// TIA Portal V17 export
// export: Created 2025-05-22T06:00:28.3771667Z, ExportSetting WithDefaults, DisplayName Totally Integrated Automation Portal, DisplayVersion V17 Update 8, DisplayName TIA Portal Openness, DisplayVersion V17 Update 8, DisplayName TIA Portal Version Control Interface, DisplayVersion V17, DisplayName SINAMICS Startdrive Advanced, DisplayVersion V17 SP2, DisplayName SINAMICS Startdrive G110M, G120, G120C, G120D, G120P, G115D, DisplayVersion V17 SP2, DisplayName SINAMICS Startdrive G130, G150, S120, S150, SINAMICS MV, S210, DisplayVersion V17 SP2, DisplayName STEP 7 Professional, DisplayVersion V17 Update 8, DisplayName SINUMERIK ONE STEP 7 Toolbox, DisplayVersion V17 Update 12, DisplayName SINUMERIK ONE PLC Basic Program Plus, DisplayVersion V17 Update 12, DisplayName SINUMERIK 840D sl STEP 7 Toolbox, DisplayVersion V17 Update 12, DisplayName STEP 7 Safety, DisplayVersion V17 Update 6, DisplayName WinCC Advanced, DisplayVersion V17 Update 8
FUNCTION "FC1401_UTILITY_SKIDS" : Void   // FC1401, LAD
{ S7_Optimized_Access := 'TRUE' }
VERSION : 0.1
// stored: AutoNumber false, IsIECCheckEnabled false, SetENOAutomatically false, UDAEnableTagReadback false
   VAR CONSTANT
      FC_NUMBER : DInt := 1401;
   END_VAR
   VAR_TEMP   // added for the SCL form of the ladder/FBD networks
      _w1 : Bool;
      _w2 : Bool;
   END_VAR
BEGIN

REGION Network 1: <<<<<<<<<<<<<<<<<<<< PNEUMATIC SYSTEM >>>>>>>>>>>>>>>>>>>>
END_REGION

REGION Network 2: CALL FB1401 PNEUMATIC SYSTEM
   // 2#0000_0001 OPTIONS 0 BIT 0 PRESSURE PRESENT OPTION
   // 2#0000_0010 OPTIONS 0 BIT 1 CONNECTION SENSOR 1 OPTION
   // 2#0000_0100 OPTIONS 0 BIT 2 CONNECTION SENSOR 2 OPTION
   // 2#0000_1000 OPTIONS 0 BIT 3 DRIVE UNBLOCKED OPTION
   // 2#0001_0000 OPTIONS 0 BIT 4 PRESSURIZED OPTION
   // 2#0010_0000 OPTIONS 0 BIT 5 UNIT 01 GRIPPER PRESSURIZED OPTION
   // 2#0100_0000 OPTIONS 0 BIT 6 UNIT 01 LABERINT PRESSURIZED OPTION
   // 2#1000_0000 OPTIONS 0 BIT 7 UNIT 01 UPPER TABLE PRESSURIZED OPTION
   // 
   // 2#0000_0001 OPTIONS 1 BIT 0 UNIT 01 LOWER TABLE PRESSURIZED OPTION
   // 2#0000_0010 OPTIONS 1 BIT 1 UNIT 01 AXIS X CART PRESSURIZED OPTION
   // 2#0000_0100 OPTIONS 1 BIT 2 UNIT 01 STATION 3 MEASURMENT UNIT PRESSURIZED OPTION
   // 2#0000_1000 OPTIONS 1 BIT 3 UNIT 01 STATION 4 MEASURMENT UNIT PRESSURIZED OPTION
   // 2#0001_0000 OPTIONS 1 BIT 4 UNIT 02 GRIPPER PRESSURIZEDPRESSURIZED OPTION
   // 2#0010_0000 OPTIONS 1 BIT 5 UNIT 02 LABERINT PRESSURIZED OPTION
   // 2#0100_0000 OPTIONS 1 BIT 6 UNIT 02 UPPER TABLE PRESSURIZED OPTION
   // 2#1000_0000 OPTIONS 1 BIT 7 UNIT 02 LOWER TABLE PRESSURIZED OPTION
   // 
   // 2#0000_0001 OPTIONS 2 BIT 0 UNIT 02 AXIS X CART PRESSURIZED OPTION
   // 2#0000_0010 OPTIONS 2 BIT 1 UNIT 02 STATION 3 MEASURMENT UNIT PRESSURIZED OPTION
   // 2#0000_0100 OPTIONS 2 BIT 2 UNIT 02 STATION 4 MEASURMENT UNIT PRESSURIZED OPTION
   // 2#0000_1000 OPTIONS 2 BIT 3 INPUT FLOW  OPTION
   // 2#0001_0000 OPTIONS 2 BIT 4 INPUT TEMPERATURE OPTION
   // 2#0010_0000 OPTIONS 2 BIT 5 SPARE OPTION
   // 2#0100_0000 OPTIONS 2 BIT 6 SPARE OPTION
   // 2#1000_0000 OPTIONS 2 BIT 7 SPARE OPTION
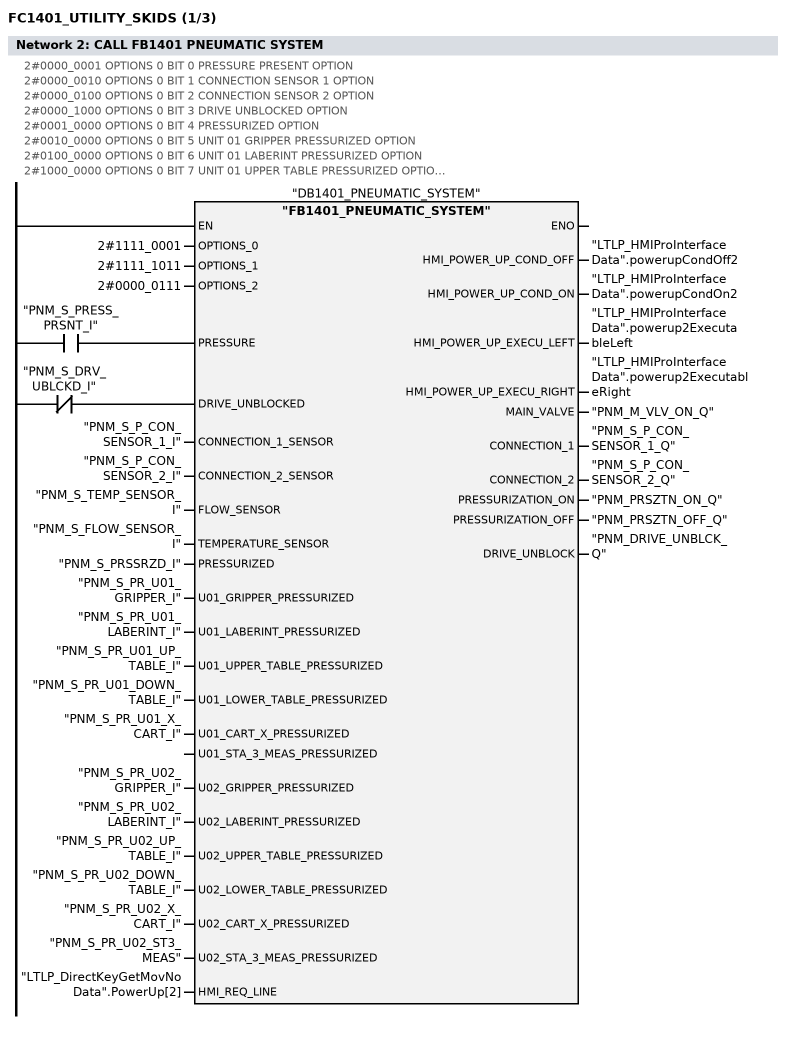
   RUNG wire#powerrail
      "DB1401_PNEUMATIC_SYSTEM"(PRESSURE := wire#w1, DRIVE_UNBLOCKED := wire#w2, OPTIONS_0 := 2#1111_0001, OPTIONS_1 := 2#1111_1011, OPTIONS_2 := 2#0000_0111, CONNECTION_1_SENSOR := "PNM_S_P_CON_SENSOR_1_I", CONNECTION_2_SENSOR := "PNM_S_P_CON_SENSOR_2_I", FLOW_SENSOR := "PNM_S_TEMP_SENSOR_I", TEMPERATURE_SENSOR := "PNM_S_FLOW_SENSOR_I", PRESSURIZED := "PNM_S_PRSSRZD_I", U01_GRIPPER_PRESSURIZED := "PNM_S_PR_U01_GRIPPER_I", U01_LABERINT_PRESSURIZED := "PNM_S_PR_U01_LABERINT_I", U01_UPPER_TABLE_PRESSURIZED := "PNM_S_PR_U01_UP_TABLE_I", U01_LOWER_TABLE_PRESSURIZED := "PNM_S_PR_U01_DOWN_TABLE_I", U01_CART_X_PRESSURIZED := "PNM_S_PR_U01_X_CART_I", U01_STA_3_MEAS_PRESSURIZED :=, U02_GRIPPER_PRESSURIZED := "PNM_S_PR_U02_GRIPPER_I", U02_LABERINT_PRESSURIZED := "PNM_S_PR_U02_LABERINT_I", U02_UPPER_TABLE_PRESSURIZED := "PNM_S_PR_U02_UP_TABLE_I", U02_LOWER_TABLE_PRESSURIZED := "PNM_S_PR_U02_DOWN_TABLE_I", U02_CART_X_PRESSURIZED := "PNM_S_PR_U02_X_CART_I", U02_STA_3_MEAS_PRESSURIZED := "PNM_S_PR_U02_ST3_MEAS", HMI_REQ_LINE := "LTLP_DirectKeyGetMovNoData".PowerUp[2], HMI_POWER_UP_COND_OFF => "LTLP_HMIProInterfaceData".powerupCondOff2, HMI_POWER_UP_COND_ON => "LTLP_HMIProInterfaceData".powerupCondOn2, HMI_POWER_UP_EXECU_LEFT => "LTLP_HMIProInterfaceData".powerup2ExecutableLeft, HMI_POWER_UP_EXECU_RIGHT => "LTLP_HMIProInterfaceData".powerup2ExecutableRight, MAIN_VALVE => "PNM_M_VLV_ON_Q", CONNECTION_1 => "PNM_S_P_CON_SENSOR_1_Q", CONNECTION_2 => "PNM_S_P_CON_SENSOR_2_Q", PRESSURIZATION_ON => "PNM_PRSZTN_ON_Q", PRESSURIZATION_OFF => "PNM_PRSZTN_OFF_Q", DRIVE_UNBLOCK => "PNM_DRIVE_UNBLCK_Q")
   END_RUNG
   RUNG wire#powerrail
      Contact( "PNM_S_PRESS_PRSNT_I" )
   END_RUNG wire#w1
   RUNG wire#powerrail
      I_Contact( "PNM_S_DRV_UBLCKD_I" )
   END_RUNG wire#w2
   // the same network as SCL:
   "DB1401_PNEUMATIC_SYSTEM"(OPTIONS_0 := 2#1111_0001,   // "FB1401_PNEUMATIC_SYSTEM"
                           OPTIONS_1 := 2#1111_1011,
                           OPTIONS_2 := 2#0000_0111,
                           PRESSURE := "PNM_S_PRESS_PRSNT_I",
                           DRIVE_UNBLOCKED := NOT "PNM_S_DRV_UBLCKD_I",
                           CONNECTION_1_SENSOR := "PNM_S_P_CON_SENSOR_1_I",
                           CONNECTION_2_SENSOR := "PNM_S_P_CON_SENSOR_2_I",
                           FLOW_SENSOR := "PNM_S_TEMP_SENSOR_I",
                           TEMPERATURE_SENSOR := "PNM_S_FLOW_SENSOR_I",
                           PRESSURIZED := "PNM_S_PRSSRZD_I",
                           U01_GRIPPER_PRESSURIZED := "PNM_S_PR_U01_GRIPPER_I",
                           U01_LABERINT_PRESSURIZED := "PNM_S_PR_U01_LABERINT_I",
                           U01_UPPER_TABLE_PRESSURIZED := "PNM_S_PR_U01_UP_TABLE_I",
                           U01_LOWER_TABLE_PRESSURIZED := "PNM_S_PR_U01_DOWN_TABLE_I",
                           U01_CART_X_PRESSURIZED := "PNM_S_PR_U01_X_CART_I",
                           U02_GRIPPER_PRESSURIZED := "PNM_S_PR_U02_GRIPPER_I",
                           U02_LABERINT_PRESSURIZED := "PNM_S_PR_U02_LABERINT_I",
                           U02_UPPER_TABLE_PRESSURIZED := "PNM_S_PR_U02_UP_TABLE_I",
                           U02_LOWER_TABLE_PRESSURIZED := "PNM_S_PR_U02_DOWN_TABLE_I",
                           U02_CART_X_PRESSURIZED := "PNM_S_PR_U02_X_CART_I",
                           U02_STA_3_MEAS_PRESSURIZED := "PNM_S_PR_U02_ST3_MEAS",
                           HMI_REQ_LINE := "LTLP_DirectKeyGetMovNoData".PowerUp[2],
                           HMI_POWER_UP_COND_OFF => "LTLP_HMIProInterfaceData".powerupCondOff2,
                           HMI_POWER_UP_COND_ON => "LTLP_HMIProInterfaceData".powerupCondOn2,
                           HMI_POWER_UP_EXECU_LEFT => "LTLP_HMIProInterfaceData".powerup2ExecutableLeft,
                           HMI_POWER_UP_EXECU_RIGHT => "LTLP_HMIProInterfaceData".powerup2ExecutableRight,
                           MAIN_VALVE => "PNM_M_VLV_ON_Q",
                           CONNECTION_1 => "PNM_S_P_CON_SENSOR_1_Q",
                           CONNECTION_2 => "PNM_S_P_CON_SENSOR_2_Q",
                           PRESSURIZATION_ON => "PNM_PRSZTN_ON_Q",
                           PRESSURIZATION_OFF => "PNM_PRSZTN_OFF_Q",
                           DRIVE_UNBLOCK => "PNM_DRIVE_UNBLCK_Q");
END_REGION

REGION Network 3: <<<<<<<<<<<<<<<<<<<< LUBRICATION SYSTEM >>>>>>>>>>>>>>>>>>>>
END_REGION

REGION Network 4: CALL FB1421 PROGRESSIVE LUBRICATION WITH GREASE
   // 2#0000_0001 OPTIONS 0 BIT 0 CIRCUIT BREAKER OPTION
   // 2#0000_0010 OPTIONS 0 BIT 1 LOW LEVEL ALARM OPTION
   // 2#0000_0100 OPTIONS 0 BIT 2 OVERPRESSURE ALARM OPTION
   // 2#0000_1000 OPTIONS 0 BIT 3 LUBRICATION BY TIME VALVE 1 AXIS X OPTION
   // 2#0001_0000 OPTIONS 0 BIT 4 LUBRICATION BY TIME VALVE 2 AXIS Z OPTION
   // 2#0010_0000 OPTIONS 0 BIT 5 LUBRICATION BY TIME VALVE 3 TURN UNIT OPTION
   // 2#0100_0000 OPTIONS 0 BIT 6 LUBRICATION BY TIME VALVE 4 OPTION
   // 2#1000_0000 OPTIONS 0 BIT 7 LUBRICATION DONE VALVE 1  AXIS X OPTION
   // 
   // 2#0000_0001 OPTIONS 1 BIT 0 LUBRICATION DONE VALVE 2 AXIS Z OPTION
   // 2#0000_0010 OPTIONS 1 BIT 1 LUBRICATION DONE VALVE 3 TURN UNIT OPTION
   // 2#0000_0100 OPTIONS 1 BIT 2 LUBRICATION DONE VALVE 4 OPTION
   // 2#0000_1000 OPTIONS 1 BIT 3 LUBRICATION DONE VALVE 5 OPTION
   // 2#0001_0000 OPTIONS 1 BIT 4 LUBRICATION DONE VALVE 6 OPTION
   // 2#0010_0000 OPTIONS 1 BIT 5 LUBRICATION DONE VALVE 7 OPTION
   // 2#0100_0000 OPTIONS 1 BIT 6 LUBRICATION DONE VALVE 8 OPTION
   // 2#1000_0000 OPTIONS 1 BIT 7 LUBRICATION DONE VALVE 9 OPTION
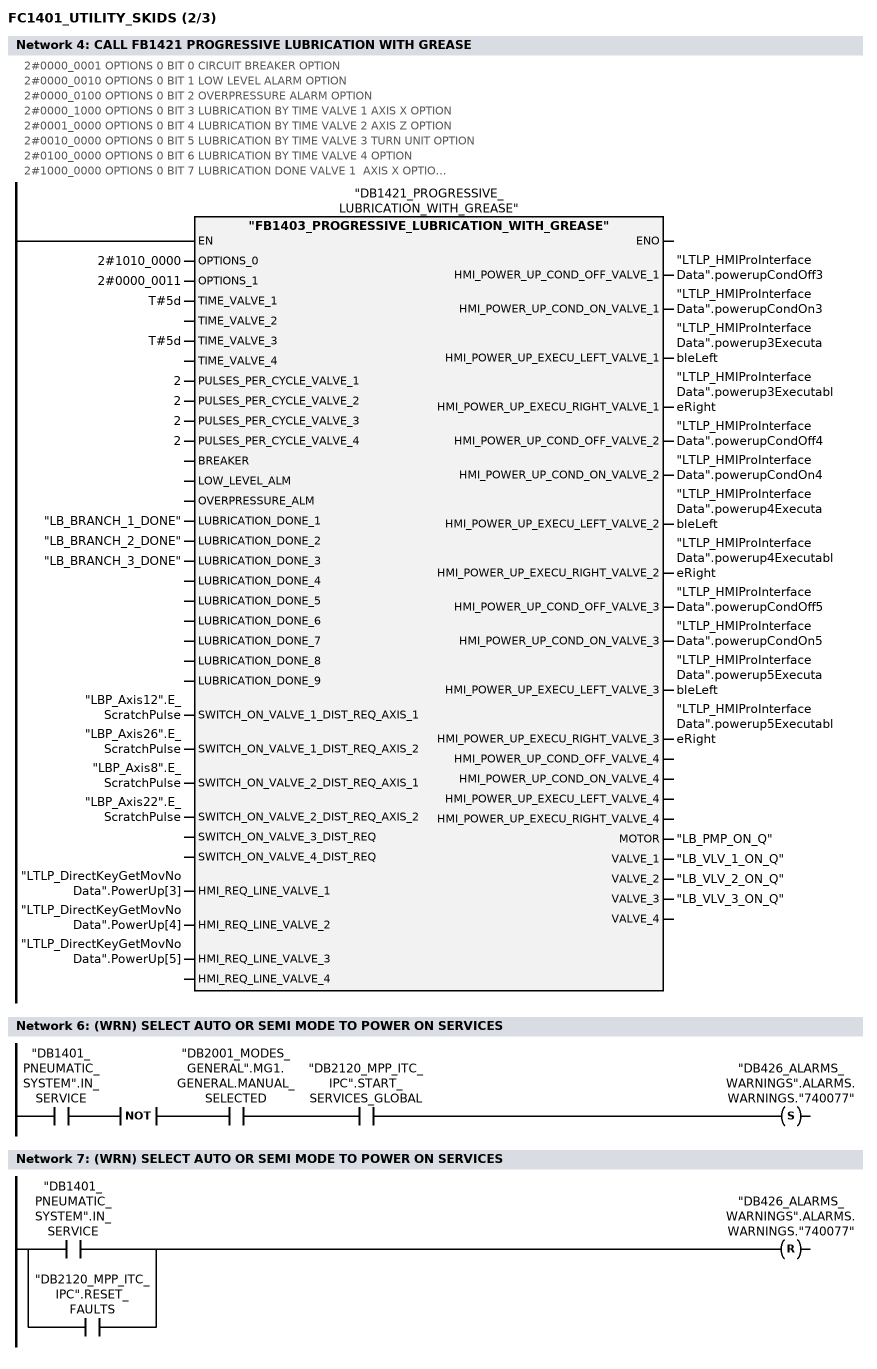
   RUNG wire#powerrail
      "DB1421_PROGRESSIVE_LUBRICATION_WITH_GREASE"(OPTIONS_0 := 2#1010_0000, OPTIONS_1 := 2#0000_0011, TIME_VALVE_1 := T#5d, TIME_VALVE_2 :=, TIME_VALVE_3 := T#5d, TIME_VALVE_4 :=, PULSES_PER_CYCLE_VALVE_1 := 2, PULSES_PER_CYCLE_VALVE_2 := 2, PULSES_PER_CYCLE_VALVE_3 := 2, PULSES_PER_CYCLE_VALVE_4 := 2, BREAKER :=, LOW_LEVEL_ALM :=, OVERPRESSURE_ALM :=, LUBRICATION_DONE_1 := "LB_BRANCH_1_DONE", LUBRICATION_DONE_2 := "LB_BRANCH_2_DONE", LUBRICATION_DONE_3 := "LB_BRANCH_3_DONE", LUBRICATION_DONE_4 :=, LUBRICATION_DONE_5 :=, LUBRICATION_DONE_6 :=, LUBRICATION_DONE_7 :=, LUBRICATION_DONE_8 :=, LUBRICATION_DONE_9 :=, SWITCH_ON_VALVE_1_DIST_REQ_AXIS_1 := "LBP_Axis12".E_ScratchPulse, SWITCH_ON_VALVE_1_DIST_REQ_AXIS_2 := "LBP_Axis26".E_ScratchPulse, SWITCH_ON_VALVE_2_DIST_REQ_AXIS_1 := "LBP_Axis8".E_ScratchPulse, SWITCH_ON_VALVE_2_DIST_REQ_AXIS_2 := "LBP_Axis22".E_ScratchPulse, SWITCH_ON_VALVE_3_DIST_REQ :=, SWITCH_ON_VALVE_4_DIST_REQ :=, HMI_REQ_LINE_VALVE_1 := "LTLP_DirectKeyGetMovNoData".PowerUp[3], HMI_REQ_LINE_VALVE_2 := "LTLP_DirectKeyGetMovNoData".PowerUp[4], HMI_REQ_LINE_VALVE_3 := "LTLP_DirectKeyGetMovNoData".PowerUp[5], HMI_REQ_LINE_VALVE_4 :=, HMI_POWER_UP_COND_OFF_VALVE_1 => "LTLP_HMIProInterfaceData".powerupCondOff3, HMI_POWER_UP_COND_ON_VALVE_1 => "LTLP_HMIProInterfaceData".powerupCondOn3, HMI_POWER_UP_EXECU_LEFT_VALVE_1 => "LTLP_HMIProInterfaceData".powerup3ExecutableLeft, HMI_POWER_UP_EXECU_RIGHT_VALVE_1 => "LTLP_HMIProInterfaceData".powerup3ExecutableRight, HMI_POWER_UP_COND_OFF_VALVE_2 => "LTLP_HMIProInterfaceData".powerupCondOff4, HMI_POWER_UP_COND_ON_VALVE_2 => "LTLP_HMIProInterfaceData".powerupCondOn4, HMI_POWER_UP_EXECU_LEFT_VALVE_2 => "LTLP_HMIProInterfaceData".powerup4ExecutableLeft, HMI_POWER_UP_EXECU_RIGHT_VALVE_2 => "LTLP_HMIProInterfaceData".powerup4ExecutableRight, HMI_POWER_UP_COND_OFF_VALVE_3 => "LTLP_HMIProInterfaceData".powerupCondOff5, HMI_POWER_UP_COND_ON_VALVE_3 => "LTLP_HMIProInterfaceData".powerupCondOn5, HMI_POWER_UP_EXECU_LEFT_VALVE_3 => "LTLP_HMIProInterfaceData".powerup5ExecutableLeft, HMI_POWER_UP_EXECU_RIGHT_VALVE_3 => "LTLP_HMIProInterfaceData".powerup5ExecutableRight, HMI_POWER_UP_COND_OFF_VALVE_4 =>, HMI_POWER_UP_COND_ON_VALVE_4 =>, HMI_POWER_UP_EXECU_LEFT_VALVE_4 =>, HMI_POWER_UP_EXECU_RIGHT_VALVE_4 =>, MOTOR => "LB_PMP_ON_Q", VALVE_1 => "LB_VLV_1_ON_Q", VALVE_2 => "LB_VLV_2_ON_Q", VALVE_3 => "LB_VLV_3_ON_Q", VALVE_4 =>)
   END_RUNG
   // the same network as SCL:
   "DB1421_PROGRESSIVE_LUBRICATION_WITH_GREASE"(OPTIONS_0 := 2#1010_0000,   // "FB1403_PROGRESSIVE_LUBRICATION_WITH_GREASE"
                           OPTIONS_1 := 2#0000_0011,
                           TIME_VALVE_1 := T#5d,
                           TIME_VALVE_3 := T#5d,
                           PULSES_PER_CYCLE_VALVE_1 := 2,
                           PULSES_PER_CYCLE_VALVE_2 := 2,
                           PULSES_PER_CYCLE_VALVE_3 := 2,
                           PULSES_PER_CYCLE_VALVE_4 := 2,
                           LUBRICATION_DONE_1 := "LB_BRANCH_1_DONE",
                           LUBRICATION_DONE_2 := "LB_BRANCH_2_DONE",
                           LUBRICATION_DONE_3 := "LB_BRANCH_3_DONE",
                           SWITCH_ON_VALVE_1_DIST_REQ_AXIS_1 := "LBP_Axis12".E_ScratchPulse,
                           SWITCH_ON_VALVE_1_DIST_REQ_AXIS_2 := "LBP_Axis26".E_ScratchPulse,
                           SWITCH_ON_VALVE_2_DIST_REQ_AXIS_1 := "LBP_Axis8".E_ScratchPulse,
                           SWITCH_ON_VALVE_2_DIST_REQ_AXIS_2 := "LBP_Axis22".E_ScratchPulse,
                           HMI_REQ_LINE_VALVE_1 := "LTLP_DirectKeyGetMovNoData".PowerUp[3],
                           HMI_REQ_LINE_VALVE_2 := "LTLP_DirectKeyGetMovNoData".PowerUp[4],
                           HMI_REQ_LINE_VALVE_3 := "LTLP_DirectKeyGetMovNoData".PowerUp[5],
                           HMI_POWER_UP_COND_OFF_VALVE_1 => "LTLP_HMIProInterfaceData".powerupCondOff3,
                           HMI_POWER_UP_COND_ON_VALVE_1 => "LTLP_HMIProInterfaceData".powerupCondOn3,
                           HMI_POWER_UP_EXECU_LEFT_VALVE_1 => "LTLP_HMIProInterfaceData".powerup3ExecutableLeft,
                           HMI_POWER_UP_EXECU_RIGHT_VALVE_1 => "LTLP_HMIProInterfaceData".powerup3ExecutableRight,
                           HMI_POWER_UP_COND_OFF_VALVE_2 => "LTLP_HMIProInterfaceData".powerupCondOff4,
                           HMI_POWER_UP_COND_ON_VALVE_2 => "LTLP_HMIProInterfaceData".powerupCondOn4,
                           HMI_POWER_UP_EXECU_LEFT_VALVE_2 => "LTLP_HMIProInterfaceData".powerup4ExecutableLeft,
                           HMI_POWER_UP_EXECU_RIGHT_VALVE_2 => "LTLP_HMIProInterfaceData".powerup4ExecutableRight,
                           HMI_POWER_UP_COND_OFF_VALVE_3 => "LTLP_HMIProInterfaceData".powerupCondOff5,
                           HMI_POWER_UP_COND_ON_VALVE_3 => "LTLP_HMIProInterfaceData".powerupCondOn5,
                           HMI_POWER_UP_EXECU_LEFT_VALVE_3 => "LTLP_HMIProInterfaceData".powerup5ExecutableLeft,
                           HMI_POWER_UP_EXECU_RIGHT_VALVE_3 => "LTLP_HMIProInterfaceData".powerup5ExecutableRight,
                           MOTOR => "LB_PMP_ON_Q",
                           VALVE_1 => "LB_VLV_1_ON_Q",
                           VALVE_2 => "LB_VLV_2_ON_Q",
                           VALVE_3 => "LB_VLV_3_ON_Q");
END_REGION

REGION Network 5: <<<<<<<<<<<<<<<<<<<< GENERAL WARNINGS >>>>>>>>>>>>>>>>>>>>
END_REGION

REGION Network 6: (WRN) SELECT AUTO OR SEMI MODE TO POWER ON SERVICES
   RUNG wire#powerrail
      Contact( "DB1401_PNEUMATIC_SYSTEM".IN_SERVICE )
      Not()
      Contact( "DB2001_MODES_GENERAL".MG1.GENERAL.MANUAL_SELECTED )
      Contact( "DB2120_MPP_ITC_IPC".START_SERVICES_GLOBAL )
      S_Coil( "DB426_ALARMS_WARNINGS".ALARMS.WARNINGS."740077" )
   END_RUNG
   // the same network as SCL:
   IF NOT "DB1401_PNEUMATIC_SYSTEM".IN_SERVICE AND "DB2001_MODES_GENERAL".MG1.GENERAL.MANUAL_SELECTED AND "DB2120_MPP_ITC_IPC".START_SERVICES_GLOBAL THEN
       "DB426_ALARMS_WARNINGS".ALARMS.WARNINGS."740077" := TRUE;
   END_IF;
END_REGION

REGION Network 7: (WRN) SELECT AUTO OR SEMI MODE TO POWER ON SERVICES
   RUNG wire#powerrail
      Contact( "DB1401_PNEUMATIC_SYSTEM".IN_SERVICE )
      wire#w1
      R_Coil( "DB426_ALARMS_WARNINGS".ALARMS.WARNINGS."740077" )
   END_RUNG
   RUNG wire#powerrail
      Contact( "DB2120_MPP_ITC_IPC".RESET_FAULTS )
   END_RUNG wire#w1
   // the same network as SCL:
   IF "DB1401_PNEUMATIC_SYSTEM".IN_SERVICE OR "DB2120_MPP_ITC_IPC".RESET_FAULTS THEN
       "DB426_ALARMS_WARNINGS".ALARMS.WARNINGS."740077" := FALSE;
   END_IF;
END_REGION

REGION Network 8: WARNINGS
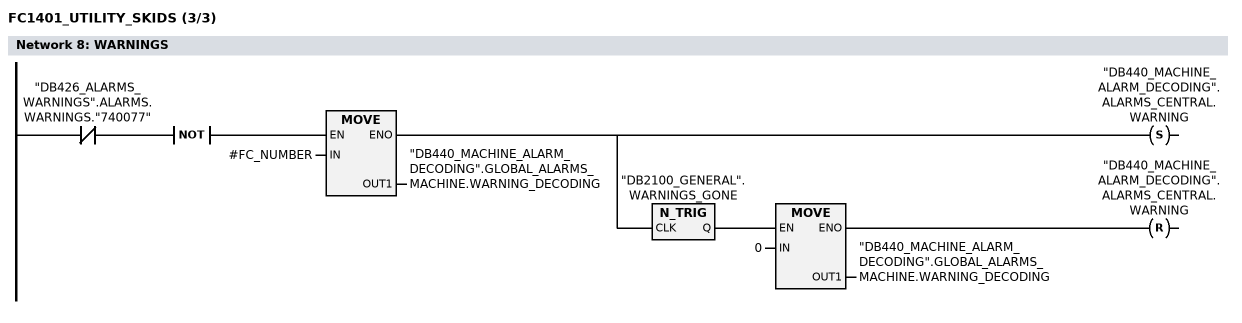
   RUNG wire#powerrail
      I_Contact( "DB426_ALARMS_WARNINGS".ALARMS.WARNINGS."740077" )
      Not()
      { S7_GenerateENO := "TRUE" } Move(in := #FC_NUMBER, out1 => "DB440_MACHINE_ALARM_DECODING".GLOBAL_ALARMS_MACHINE.WARNING_DECODING)
      wire#w1
      S_Coil( "DB440_MACHINE_ALARM_DECODING".ALARMS_CENTRAL.WARNING )
   END_RUNG
   RUNG wire#w1
      N_Trig( "DB2100_GENERAL".WARNINGS_GONE )
      { S7_GenerateENO := "TRUE" } Move(in := 0, out1 => "DB440_MACHINE_ALARM_DECODING".GLOBAL_ALARMS_MACHINE.WARNING_DECODING)
      R_Coil( "DB440_MACHINE_ALARM_DECODING".ALARMS_CENTRAL.WARNING )
   END_RUNG
   // the same network as SCL:
   // ENO of a box is taken as its EN; it also drops when the box reports an error
   #_w1 := NOT (NOT "DB426_ALARMS_WARNINGS".ALARMS.WARNINGS."740077");
   IF #_w1 THEN
       "DB440_MACHINE_ALARM_DECODING".GLOBAL_ALARMS_MACHINE.WARNING_DECODING := #FC_NUMBER;
       "DB440_MACHINE_ALARM_DECODING".ALARMS_CENTRAL.WARNING := TRUE;
   END_IF;
   #_w2 := NOT #_w1 AND "DB2100_GENERAL".WARNINGS_GONE;   // falling edge
   "DB2100_GENERAL".WARNINGS_GONE := #_w1;
   IF #_w2 THEN
       "DB440_MACHINE_ALARM_DECODING".GLOBAL_ALARMS_MACHINE.WARNING_DECODING := 0;
       "DB440_MACHINE_ALARM_DECODING".ALARMS_CENTRAL.WARNING := FALSE;
   END_IF;
END_REGION
END_FUNCTION
